PROGRAM MBUS_Zaehler (* hier wird die Klemme, an welche der M-Bus mit den Zählern angeschlossen ist, alle 10ms aufgerufen *)
VAR
	Kommunikation_Klemme: FB_MBUSKL6781;

	Stromzaehler_BHKW_321		: FB_MBUS_General_Ext;
	Stromzaehler_BHKW_322	: FB_MBUS_General_Ext;
	Stromzaehler_Buerotrakt	: FB_MBUS_General_Ext;

	Stromzaehler_Gebaeude: FB_MBUS_General_Ext;
	Stromzaehler_Halle_TGA: FB_MBUS_General_Ext;
	Stromzaehler_Halle_Licht: FB_MBUS_General_Ext;
	Gaszaehler_BHKW1: FB_MBUS_General_Ext;
	Gaszaehler_BHKW2: FB_MBUS_General_Ext;

	WZ_4371_WP_946	: FB_MBUS_General_Ext;
	WZ_4372_WP_946	: FB_MBUS_General_Ext;
	Janitza_UMG_604: FB_MBReadInputRegs;

END_VAR

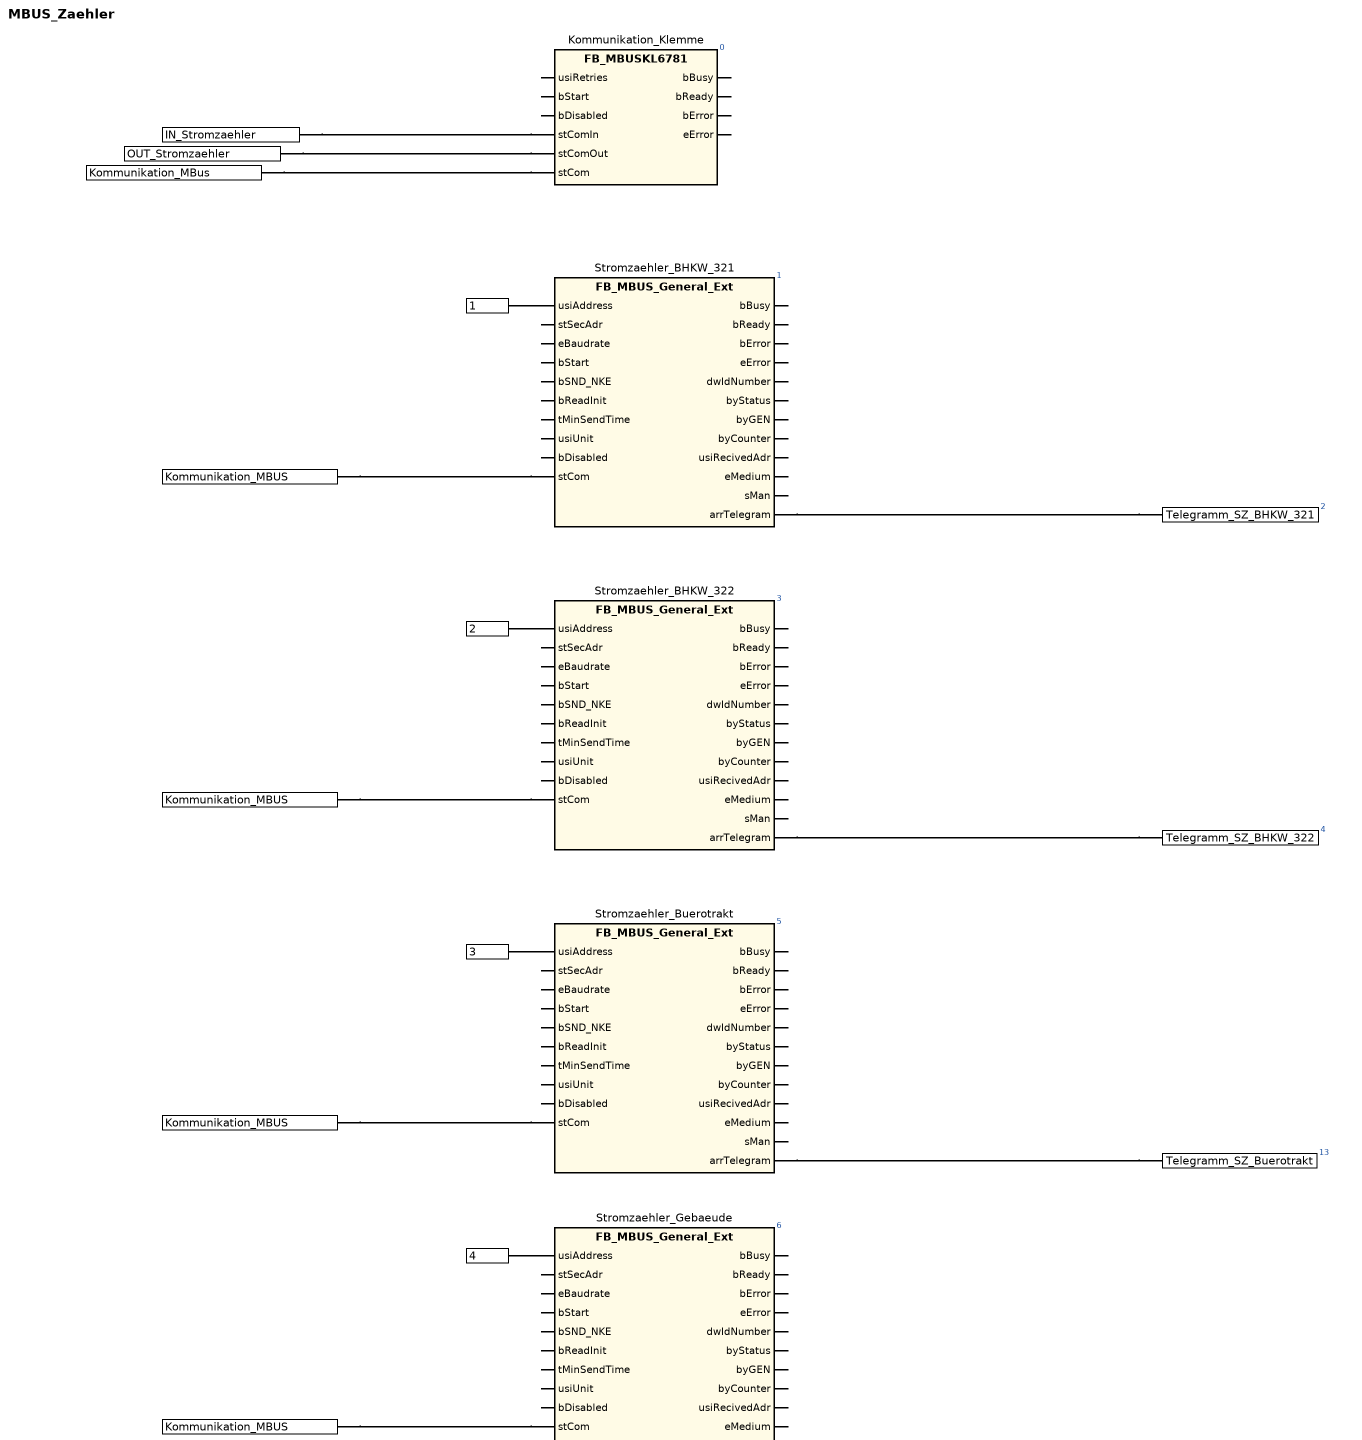
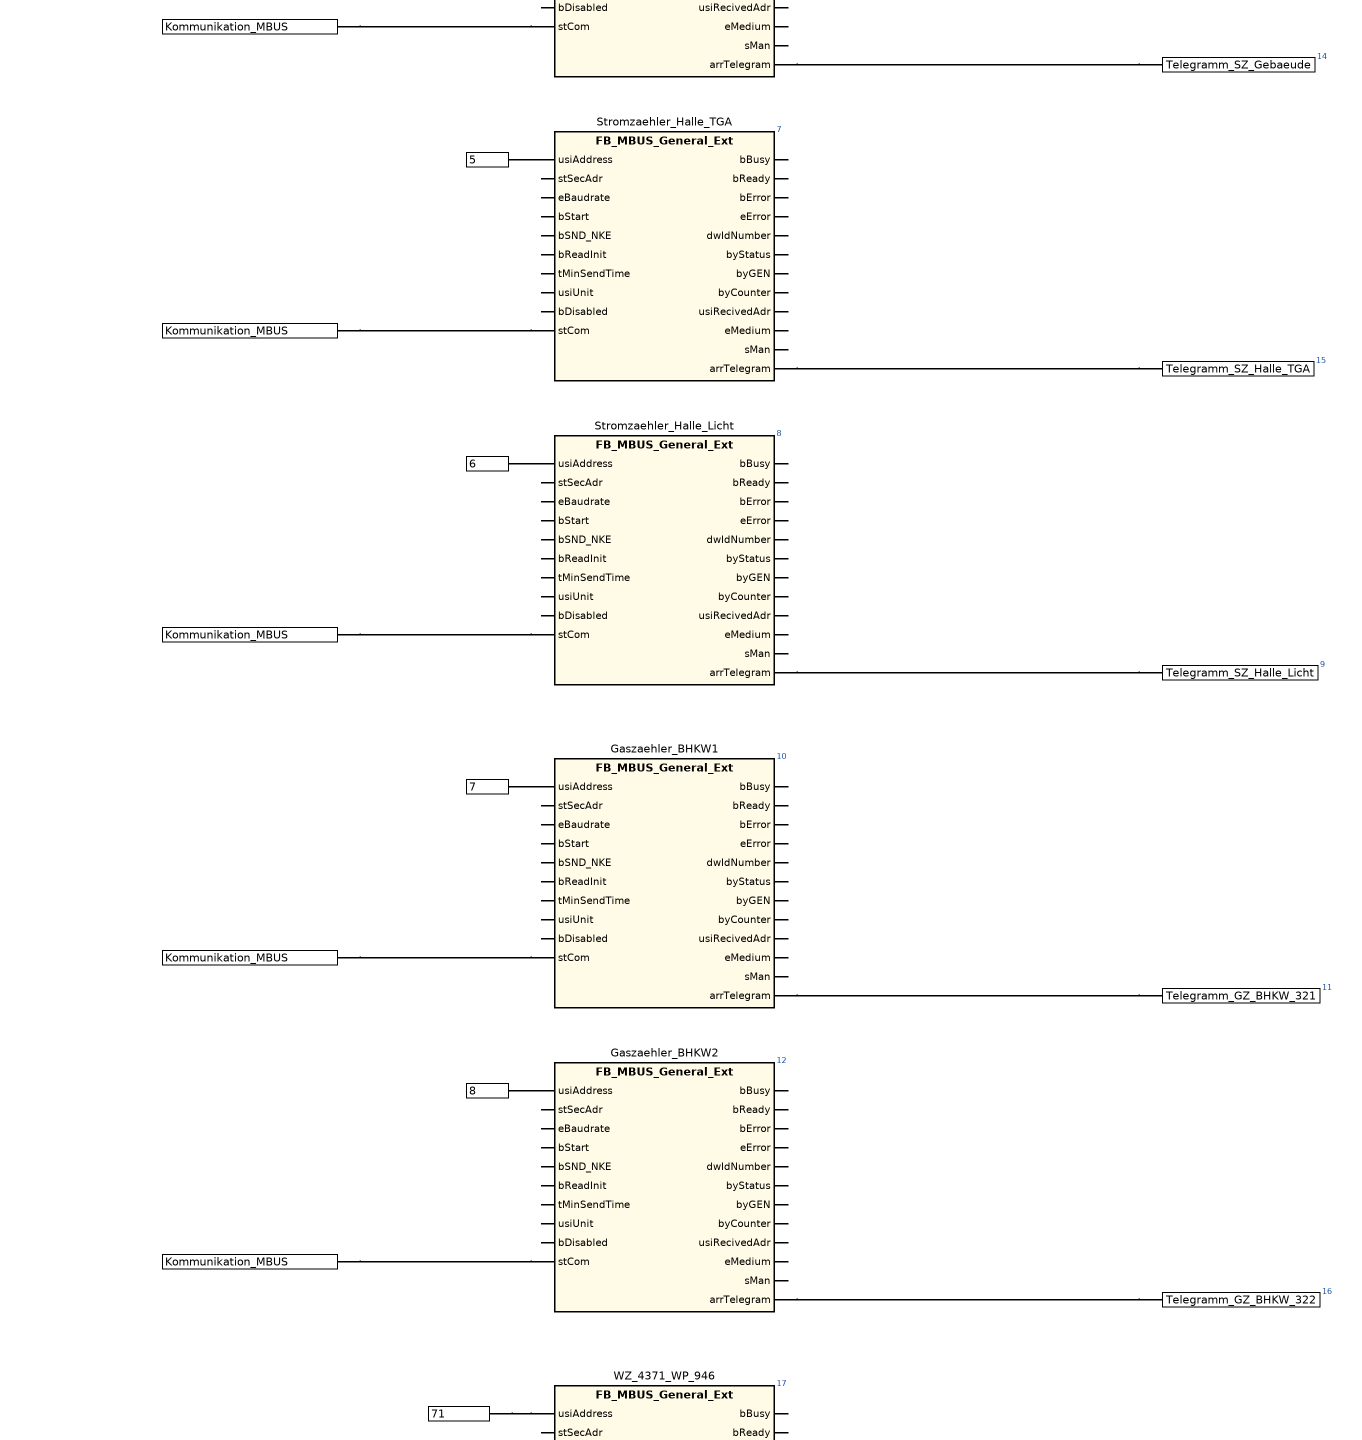
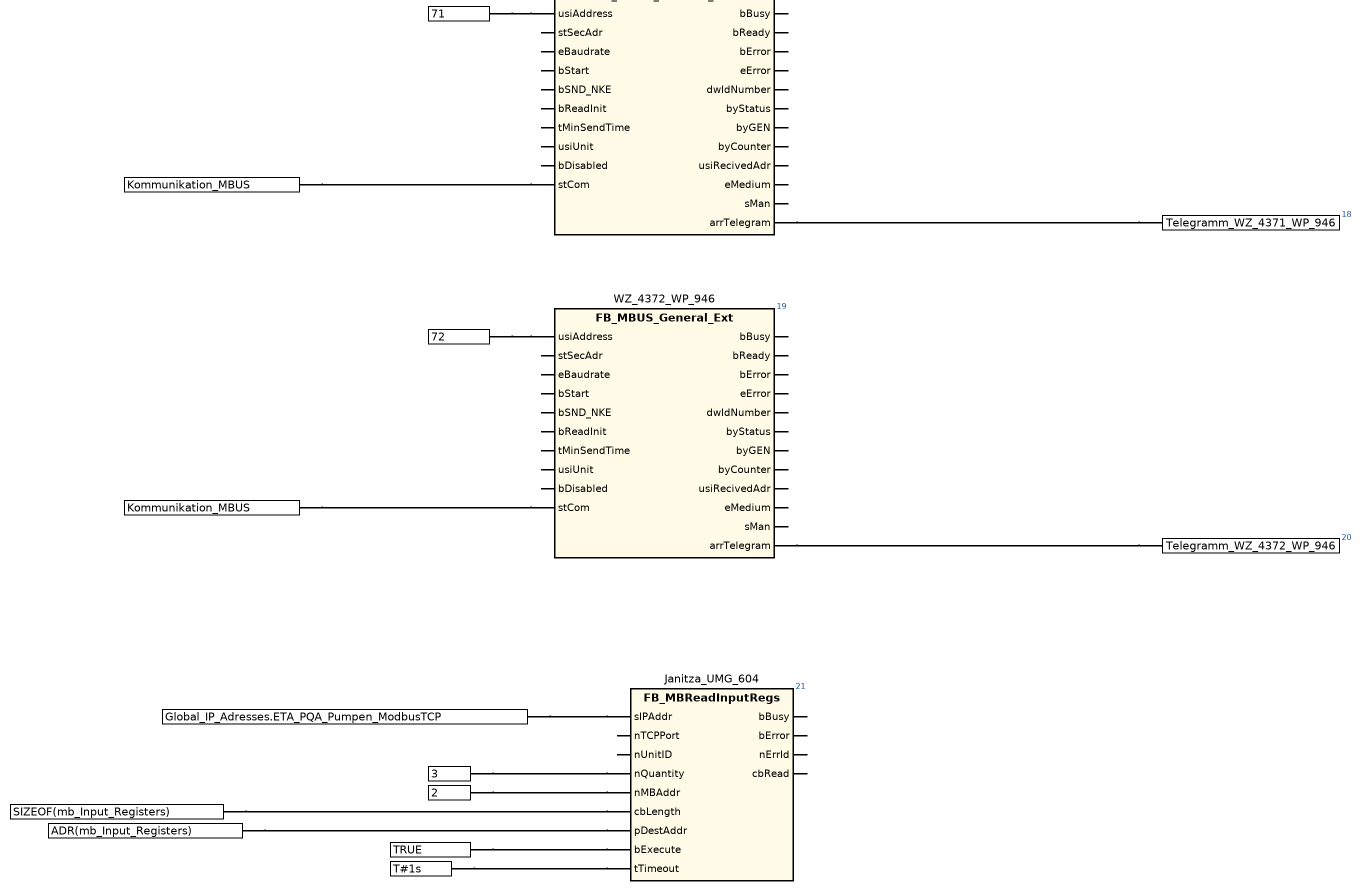
Kommunikation_Klemme(stComIn := IN_Stromzaehler, stComOut := OUT_Stromzaehler, stCom := Kommunikation_MBus); // FB_MBUSKL6781
Stromzaehler_BHKW_321(usiAddress := 1, stCom := Kommunikation_MBUS); // FB_MBUS_General_Ext
Telegramm_SZ_BHKW_321 := Stromzaehler_BHKW_321.arrTelegram;
Stromzaehler_BHKW_322(usiAddress := 2, stCom := Kommunikation_MBUS); // FB_MBUS_General_Ext
Telegramm_SZ_BHKW_322 := Stromzaehler_BHKW_322.arrTelegram;
Stromzaehler_Buerotrakt(usiAddress := 3, stCom := Kommunikation_MBUS); // FB_MBUS_General_Ext
Stromzaehler_Gebaeude(usiAddress := 4, stCom := Kommunikation_MBUS); // FB_MBUS_General_Ext
Stromzaehler_Halle_TGA(usiAddress := 5, stCom := Kommunikation_MBUS); // FB_MBUS_General_Ext
Stromzaehler_Halle_Licht(usiAddress := 6, stCom := Kommunikation_MBUS); // FB_MBUS_General_Ext
Telegramm_SZ_Halle_Licht := Stromzaehler_Halle_Licht.arrTelegram;
Gaszaehler_BHKW1(usiAddress := 7, stCom := Kommunikation_MBUS); // FB_MBUS_General_Ext
Telegramm_GZ_BHKW_321 := Gaszaehler_BHKW1.arrTelegram;
Gaszaehler_BHKW2(usiAddress := 8, stCom := Kommunikation_MBUS); // FB_MBUS_General_Ext
Telegramm_SZ_Buerotrakt := Stromzaehler_Buerotrakt.arrTelegram;
Telegramm_SZ_Gebaeude := Stromzaehler_Gebaeude.arrTelegram;
Telegramm_SZ_Halle_TGA := Stromzaehler_Halle_TGA.arrTelegram;
Telegramm_GZ_BHKW_322 := Gaszaehler_BHKW2.arrTelegram;
WZ_4371_WP_946(usiAddress := 71, stCom := Kommunikation_MBUS); // FB_MBUS_General_Ext
Telegramm_WZ_4371_WP_946 := WZ_4371_WP_946.arrTelegram;
WZ_4372_WP_946(usiAddress := 72, stCom := Kommunikation_MBUS); // FB_MBUS_General_Ext
Telegramm_WZ_4372_WP_946 := WZ_4372_WP_946.arrTelegram;
Janitza_UMG_604(
    sIPAddr := Global_IP_Adresses.ETA_PQA_Pumpen_ModbusTCP,
    nQuantity := 3,
    nMBAddr := 2,
    cbLength := SIZEOF(mb_Input_Registers),
    pDestAddr := ADR(mb_Input_Registers),
    bExecute := TRUE,
    tTimeout := T#1s); // FB_MBReadInputRegs

END_PROGRAM

(* stored: Version 1.1.0.1, ProductVersion 3.1.4024.9
   POU MBUS_Zaehler: Id {f415fce9-15f4-4c44-8ff2-ffc38c87d5d3}, SpecialFunc None *)
